(* Logix 5000 project; controller AdvManLab vendor 1 type 14 code 158 rev 28.12; software revision 28.01; part 9 of 13 *)
(* tags used below, declared in another part *)
   HMI_WritePart : DINT;
   ABB_Loop_Speed : DINT;
   Advance_Slide : BOOL;
   AutoDelay : TIMER;
   Cell1PalletAtStop : BOOL;   // Part at Cell 1 Pallet Stop
   Clamp_To_Line : BOOL;
   Close_Clamp : BOOL;
   CNC_1_Done : BOOL;   // CNC 1 has completed cutting the part
   CNC_2_Done : BOOL;   // CNC 2 has completed cutting the part
   Enable_Cell_3 : BOOL;   // Turn bit on to enable logic for Cell 3
   Enable_CNC1 : BOOL;
   Enable_CNC2 : BOOL;
   Enable_CNC3 : BOOL;
   Enable_CNC4 : BOOL;
   EnableBits : DINT;
   Extend_Stop : BOOL;
   Fanuc_Loop_Speed : DINT;
   Festo_Air_On : BOOL;
   FestoAI0 : DINT;
   FestoAI1 : DINT;
   FestoAI2 : DINT;
   FestoAI3 : DINT;
   FestoAIP0 : DINT;
   FestoAIP1 : DINT;
   FestoAIP2 : DINT;
   FestoAIP3 : DINT;
   Gantry_busy : BOOL;
   Gantry_prep : BOOL;
   Gantry_reload : BOOL;
   Gantry_start : BOOL;
   HMI_Disp_No : DINT;
   HMI_Mode : DINT;
   Lower_Slide : BOOL;
   Mode_Auto : BOOL;
   Mode_Manual : BOOL;
   Mode_None : BOOL;
   Mode_Semi : BOOL;
   Mode_Start : BOOL;
   NI_1752_Camera : MESSAGE;
   ONS : DINT;
   Open_Clamp : BOOL;
   PalletAtC2C3HoldBack : BOOL;   // Pallet at Cell 2 to Cell 3 Diverter Hold Back Stop
   Part_A : BOOL;
   Part_A_input : COUNTER;
   Part_A_output : COUNTER;
   Part_B : BOOL;
   Part_B_input : COUNTER;
   Part_B_output : COUNTER;
   Part_dropped : BOOL;
   Part_from_conv_holding : BOOL;
   Part_ready_for_Gantry : BOOL;
   Picking_up_part : BOOL;
   PPX4 : ALIAS FOR Conv_N053:3:I.2;   // Sensor Pallet Stop RFID4 (Loop 1 Diverter Hold Back Stop)
   PPX5 : ALIAS FOR Main_N043:3:I.0;   // Sensor Pallet Stop (Cell 1 Hold Back)
   R1J_Assign : BOOL;
   R1J_Check_Process_NO : DINT;
   R1J_Current_Part_NO : SINT;
   R1J_Current_Process_NO : SINT;
   R1J_Read : BOOL;
   R1J_Read_Check_Fail : BOOL;
   R1J_Read_Check_InProgress : BOOL;
   R1J_Read_Check_Results : BOOL;
   R1J_Read_Check_Start : BOOL;
   R1J_Read_Finished : BOOL;
   R1J_Read_InProgress : BOOL;
   R1J_Read_Results : BOOL;
   R1J_Read_Start : BOOL;
   R1J_Write : BOOL;
   R1J_Write_Finished_Check : BOOL;
   R1J_Write_Inprogress : BOOL;
   R1J_Write_Pass : BOOL;
   Raise_Slide : BOOL;
   Return_Slide : BOOL;
   RFID_ReadData5p : DINT;
   RFIDTP1 : ALIAS FOR RFID_N054:I.Channel[0].TagPresent;   // RFID Tag at Cell 1 Stop
   Robot1_DroppedP1 : BOOL;
   Robot1_DroppedP2 : BOOL;
   Robot1_Flipped : BOOL;
   Robot1DroppedPart : BOOL;
   Run_gantry_logic : BOOL;
   TimerG1 : TIMER;
   Vac_On : BOOL;
   Vac_To_Line : BOOL;
(* MainProgram, continued *)

ROUTINE Grantry_Logic_Prep   (* ladder *)
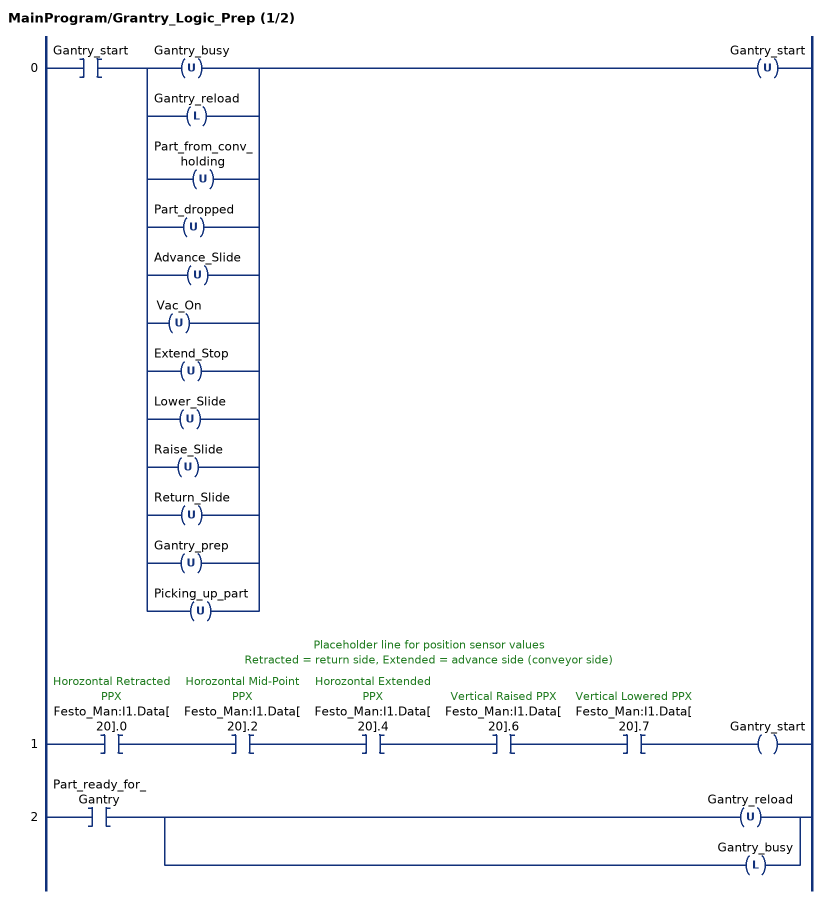
   0: XIC(Gantry_start)[OTU(Gantry_busy) ,OTL(Gantry_reload) ,OTU(Part_from_conv_holding) ,OTU(Part_dropped) ,OTU(Advance_Slide) ,OTU(Vac_On) ,OTU(Extend_Stop) ,OTU(Lower_Slide) ,OTU(Raise_Slide) ,OTU(Return_Slide) ,OTU(Gantry_prep) ,OTU(Picking_up_part) ]OTU(Gantry_start);
   // Placeholder line for position sensor values
   // Retracted = return side, Extended = advance side (conveyor side)
   1: XIC(Festo_Man:I1.Data[20].0)XIC(Festo_Man:I1.Data[20].2)XIC(Festo_Man:I1.Data[20].4)XIC(Festo_Man:I1.Data[20].6)XIC(Festo_Man:I1.Data[20].7)OTE(Gantry_start);
   2: XIC(Part_ready_for_Gantry)[OTU(Gantry_reload) ,OTL(Gantry_busy) ];
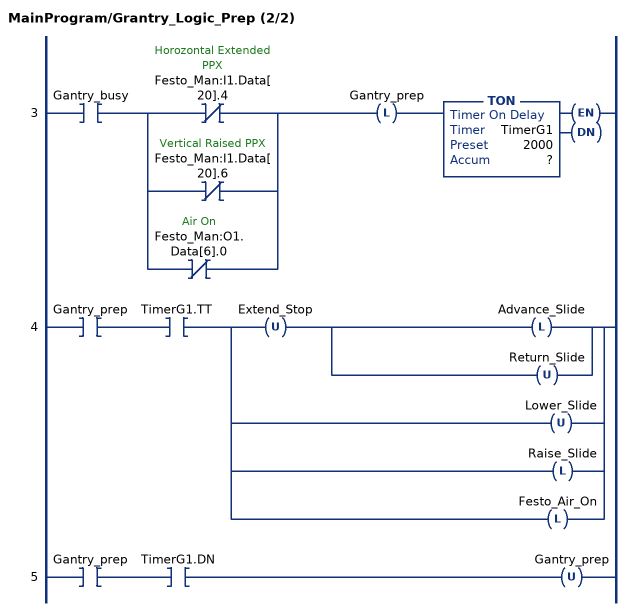
   3: XIC(Gantry_busy)[XIO(Festo_Man:I1.Data[20].4) ,XIO(Festo_Man:I1.Data[20].6) ,XIO(Festo_Man:O1.Data[6].0) ]OTL(Gantry_prep)TON(TimerG1,?,?);
   4: XIC(Gantry_prep)XIC(TimerG1.TT)[OTU(Extend_Stop) [OTL(Advance_Slide) ,OTU(Return_Slide) ] ,[OTU(Lower_Slide) ,OTL(Raise_Slide) ] ,OTL(Festo_Air_On) ];
   5: XIC(Gantry_prep)XIC(TimerG1.DN)OTU(Gantry_prep);
END_ROUTINE

ROUTINE HMI   (* ladder *)
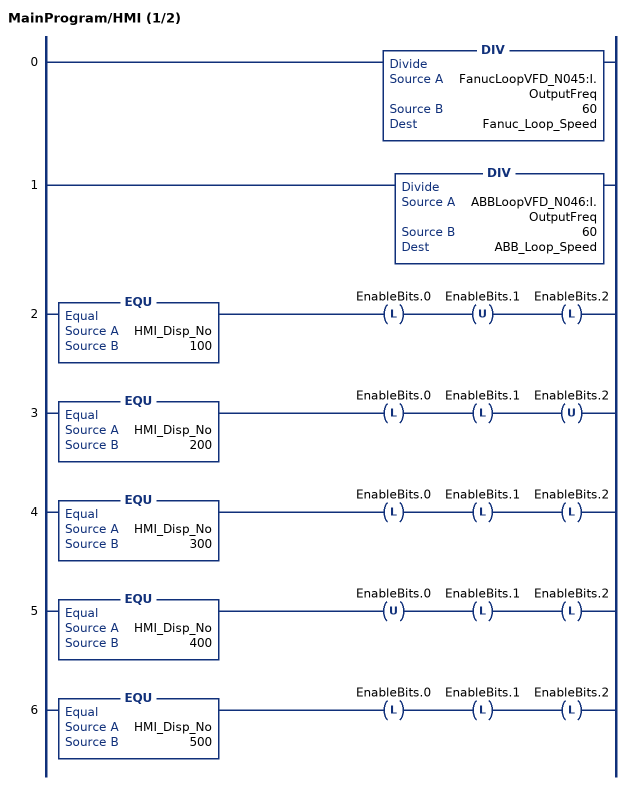
   0: DIV(FanucLoopVFD_N045:I.OutputFreq,60,Fanuc_Loop_Speed);
   1: DIV(ABBLoopVFD_N046:I.OutputFreq,60,ABB_Loop_Speed);
   2: EQU(HMI_Disp_No,100)OTL(EnableBits.0)OTU(EnableBits.1)OTL(EnableBits.2);
   3: EQU(HMI_Disp_No,200)OTL(EnableBits.0)OTL(EnableBits.1)OTU(EnableBits.2);
   4: EQU(HMI_Disp_No,300)OTL(EnableBits.0)OTL(EnableBits.1)OTL(EnableBits.2);
   5: EQU(HMI_Disp_No,400)OTU(EnableBits.0)OTL(EnableBits.1)OTL(EnableBits.2);
   6: EQU(HMI_Disp_No,500)OTL(EnableBits.0)OTL(EnableBits.1)OTL(EnableBits.2);
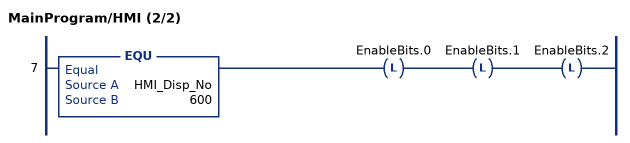
   7: EQU(HMI_Disp_No,600)OTL(EnableBits.0)OTL(EnableBits.1)OTL(EnableBits.2);
END_ROUTINE

ROUTINE MainRoutine   (* ladder *)
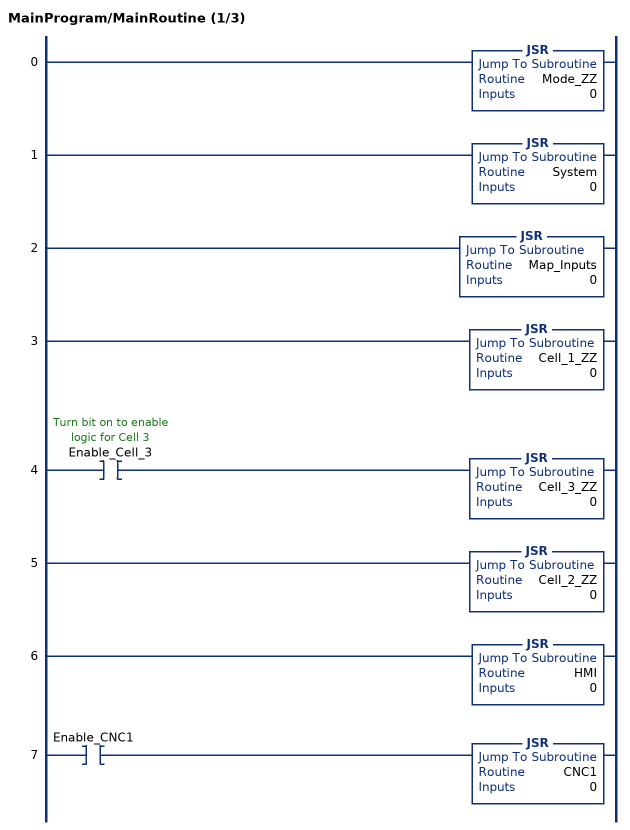
   0: JSR(Mode_ZZ,0);
   1: JSR(System,0);
   2: JSR(Map_Inputs,0);
   3: JSR(Cell_1_ZZ,0);
   4: XIC(Enable_Cell_3)JSR(Cell_3_ZZ,0);
   5: JSR(Cell_2_ZZ,0);
   6: JSR(HMI,0);
   7: XIC(Enable_CNC1)JSR(CNC1,0);
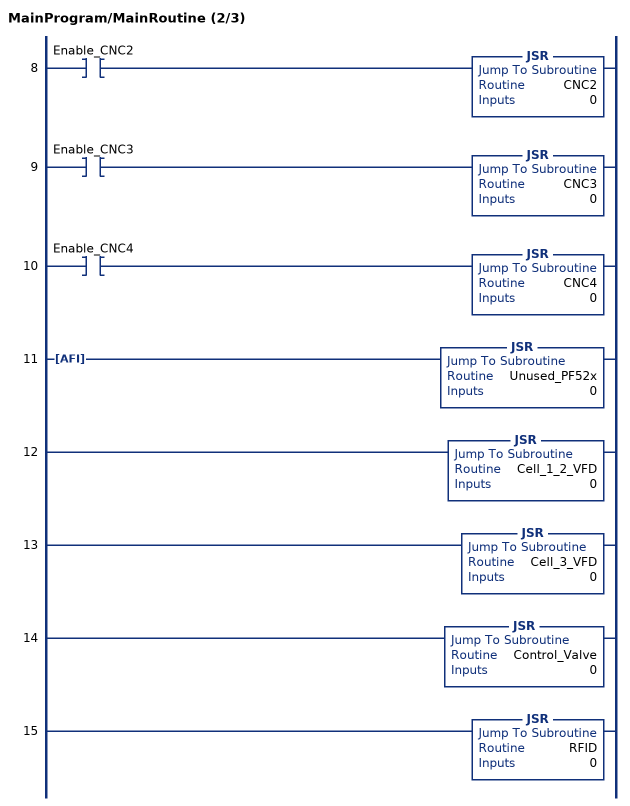
   8: XIC(Enable_CNC2)JSR(CNC2,0);
   9: XIC(Enable_CNC3)JSR(CNC3,0);
   10: XIC(Enable_CNC4)JSR(CNC4,0);
   11: AFI()JSR(Unused_PF52x,0);
   12: JSR(Cell_1_2_VFD,0);
   13: JSR(Cell_3_VFD,0);
   14: JSR(Control_Valve,0);
   15: JSR(RFID,0);
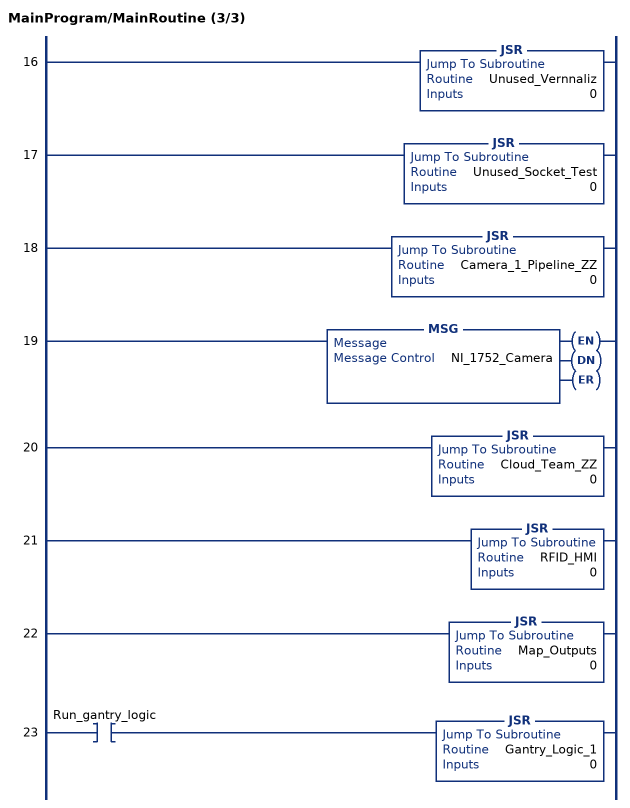
   16: JSR(Unused_Vernnaliz,0);
   17: JSR(Unused_Socket_Test,0);
   18: JSR(Camera_1_Pipeline_ZZ,0);
   19: MSG(NI_1752_Camera);
   20: JSR(Cloud_Team_ZZ,0);
   21: JSR(RFID_HMI,0);
   22: JSR(Map_Outputs,0);
   23: XIC(Run_gantry_logic)JSR(Gantry_Logic_1,0);
END_ROUTINE

ROUTINE Map_Inputs   (* ladder *)
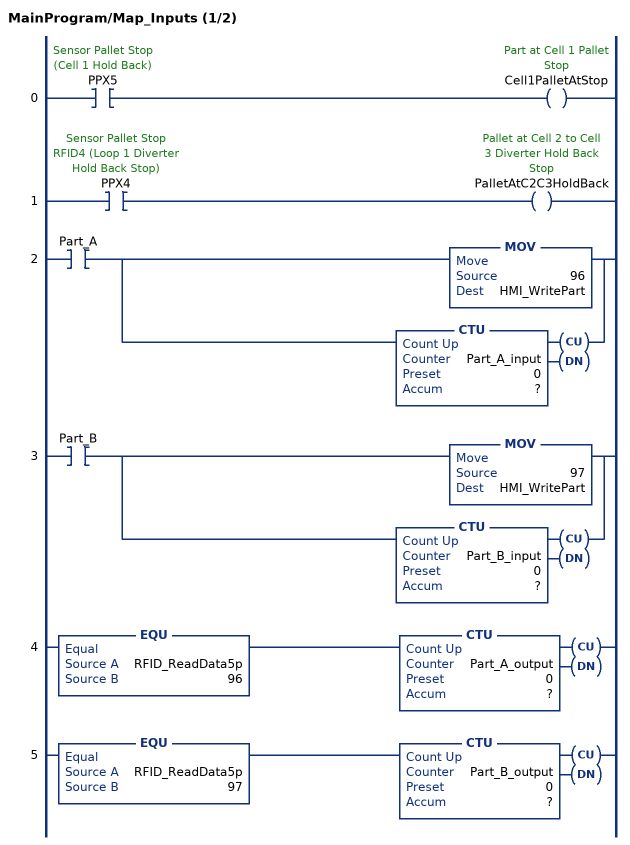
   0: XIC(PPX5)OTE(Cell1PalletAtStop);
   1: XIC(PPX4)OTE(PalletAtC2C3HoldBack);
   2: XIC(Part_A)[MOV(96,HMI_WritePart) ,CTU(Part_A_input,?,?) ];
   3: XIC(Part_B)[MOV(97,HMI_WritePart) ,CTU(Part_B_input,?,?) ];
   4: EQU(RFID_ReadData5p,96)CTU(Part_A_output,?,?);
   5: EQU(RFID_ReadData5p,97)CTU(Part_B_output,?,?);
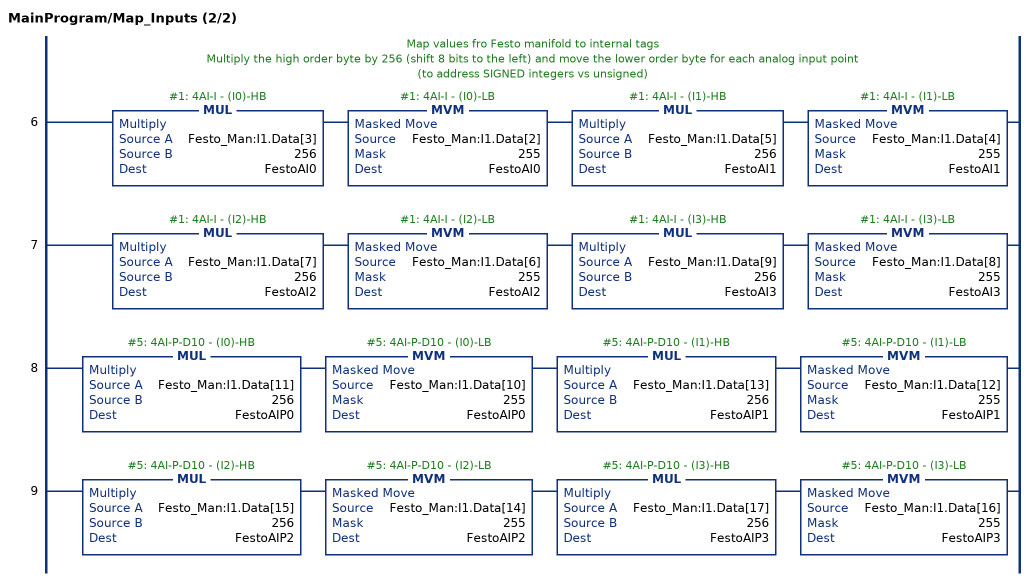
   // Map values fro Festo manifold to internal tags
   // Multiply the high order byte by 256 (shift 8 bits to the left) and move the lower order byte for each analog input point
   // (to address SIGNED integers vs unsigned)
   6: MUL(Festo_Man:I1.Data[3],256,FestoAI0)MVM(Festo_Man:I1.Data[2],255,FestoAI0)MUL(Festo_Man:I1.Data[5],256,FestoAI1)MVM(Festo_Man:I1.Data[4],255,FestoAI1);
   7: MUL(Festo_Man:I1.Data[7],256,FestoAI2)MVM(Festo_Man:I1.Data[6],255,FestoAI2)MUL(Festo_Man:I1.Data[9],256,FestoAI3)MVM(Festo_Man:I1.Data[8],255,FestoAI3);
   8: MUL(Festo_Man:I1.Data[11],256,FestoAIP0)MVM(Festo_Man:I1.Data[10],255,FestoAIP0)MUL(Festo_Man:I1.Data[13],256,FestoAIP1)MVM(Festo_Man:I1.Data[12],255,FestoAIP1);
   9: MUL(Festo_Man:I1.Data[15],256,FestoAIP2)MVM(Festo_Man:I1.Data[14],255,FestoAIP2)MUL(Festo_Man:I1.Data[17],256,FestoAIP3)MVM(Festo_Man:I1.Data[16],255,FestoAIP3);
END_ROUTINE

ROUTINE Map_Outputs   (* ladder *)
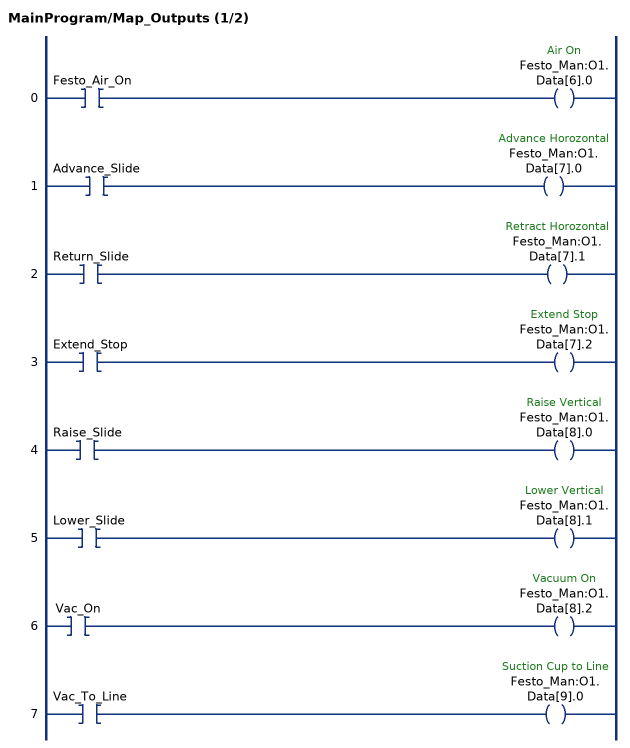
   0: XIC(Festo_Air_On)OTE(Festo_Man:O1.Data[6].0);
   1: XIC(Advance_Slide)OTE(Festo_Man:O1.Data[7].0);
   2: XIC(Return_Slide)OTE(Festo_Man:O1.Data[7].1);
   3: XIC(Extend_Stop)OTE(Festo_Man:O1.Data[7].2);
   4: XIC(Raise_Slide)OTE(Festo_Man:O1.Data[8].0);
   5: XIC(Lower_Slide)OTE(Festo_Man:O1.Data[8].1);
   6: XIC(Vac_On)OTE(Festo_Man:O1.Data[8].2);
   7: XIC(Vac_To_Line)OTE(Festo_Man:O1.Data[9].0);
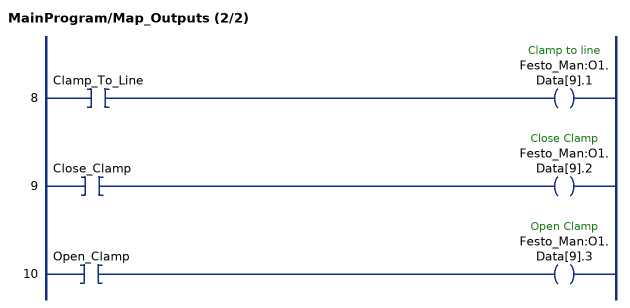
   8: XIC(Clamp_To_Line)OTE(Festo_Man:O1.Data[9].1);
   9: XIC(Close_Clamp)OTE(Festo_Man:O1.Data[9].2);
   10: XIC(Open_Clamp)OTE(Festo_Man:O1.Data[9].3);
END_ROUTINE

ROUTINE Mode_ZZ   (* ladder *)
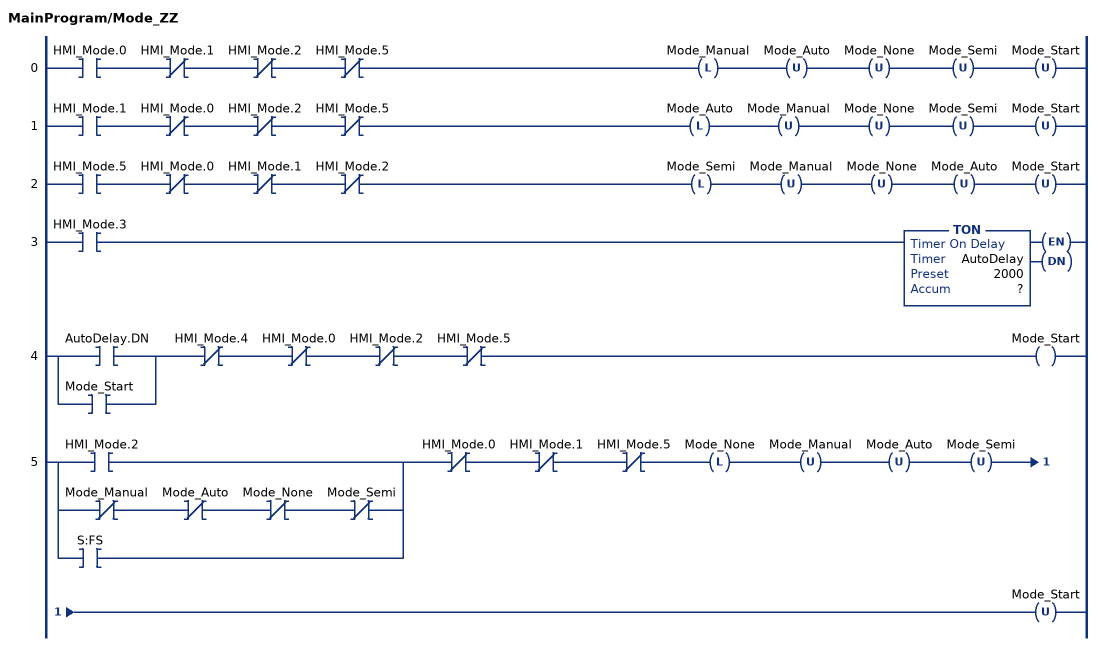
   0: XIC(HMI_Mode.0)XIO(HMI_Mode.1)XIO(HMI_Mode.2)XIO(HMI_Mode.5)OTL(Mode_Manual)OTU(Mode_Auto)OTU(Mode_None)OTU(Mode_Semi)OTU(Mode_Start);
   1: XIC(HMI_Mode.1)XIO(HMI_Mode.0)XIO(HMI_Mode.2)XIO(HMI_Mode.5)OTL(Mode_Auto)OTU(Mode_Manual)OTU(Mode_None)OTU(Mode_Semi)OTU(Mode_Start);
   2: XIC(HMI_Mode.5)XIO(HMI_Mode.0)XIO(HMI_Mode.1)XIO(HMI_Mode.2)OTL(Mode_Semi)OTU(Mode_Manual)OTU(Mode_None)OTU(Mode_Auto)OTU(Mode_Start);
   3: XIC(HMI_Mode.3)TON(AutoDelay,?,?);
   4: [XIC(AutoDelay.DN) ,XIC(Mode_Start) ]XIO(HMI_Mode.4)XIO(HMI_Mode.0)XIO(HMI_Mode.2)XIO(HMI_Mode.5)OTE(Mode_Start);
   5: [XIC(HMI_Mode.2) ,XIO(Mode_Manual) XIO(Mode_Auto) XIO(Mode_None) XIO(Mode_Semi) ,XIC(S:FS) ]XIO(HMI_Mode.0)XIO(HMI_Mode.1)XIO(HMI_Mode.5)OTL(Mode_None)OTU(Mode_Manual)OTU(Mode_Auto)OTU(Mode_Semi)OTU(Mode_Start);
END_ROUTINE

ROUTINE RFID   (* ladder *)
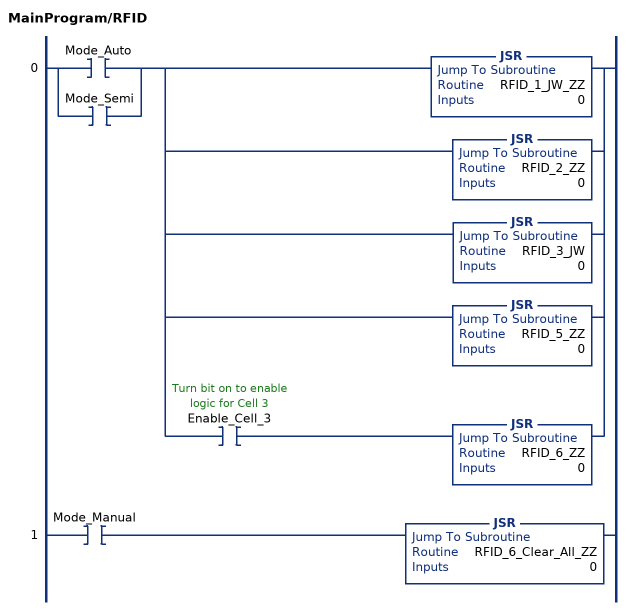
   0: [XIC(Mode_Auto) ,XIC(Mode_Semi) ][JSR(RFID_1_JW_ZZ,0) ,JSR(RFID_2_ZZ,0) ,JSR(RFID_3_JW,0) ,JSR(RFID_5_ZZ,0) ,XIC(Enable_Cell_3) JSR(RFID_6_ZZ,0) ];
   1: XIC(Mode_Manual)JSR(RFID_6_Clear_All_ZZ,0);
END_ROUTINE

ROUTINE RFID_1_JW_ZZ   (* ladder *)
// Rewrite of RFID_1 using new read/write logic of RFID_6_ZZ
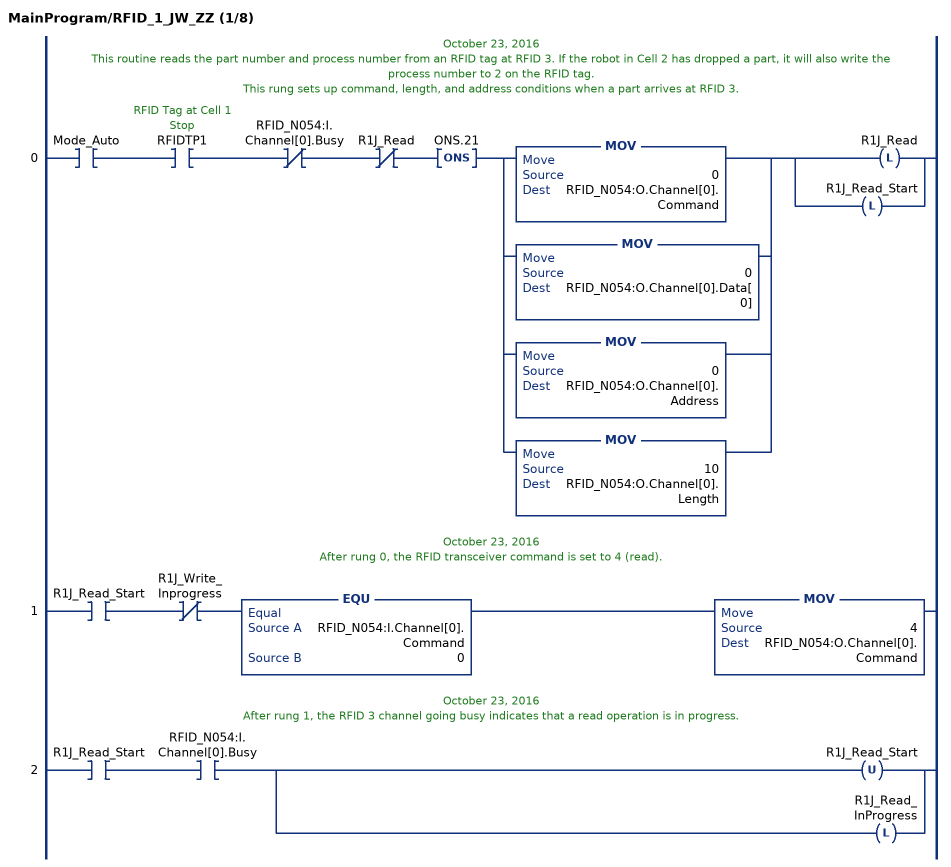
   // October 23, 2016
   // This routine reads the part number and process number from an RFID tag at RFID 3. If the robot in Cell 2 has dropped a part, it will also write the process number to 2 on the RFID tag.
   // This rung sets up command, length, and address conditions when a part arrives at RFID 3.
   0: XIC(Mode_Auto)XIC(RFIDTP1)XIO(RFID_N054:I.Channel[0].Busy)XIO(R1J_Read)ONS(ONS.21)[MOV(0,RFID_N054:O.Channel[0].Command) ,MOV(0,RFID_N054:O.Channel[0].Data[0]) ,MOV(0,RFID_N054:O.Channel[0].Address) ,MOV(10,RFID_N054:O.Channel[0].Length) ][OTL(R1J_Read) ,OTL(R1J_Read_Start) ];
   // October 23, 2016
   // After rung 0, the RFID transceiver command is set to 4 (read).
   1: XIC(R1J_Read_Start)XIO(R1J_Write_Inprogress)EQU(RFID_N054:I.Channel[0].Command,0)MOV(4,RFID_N054:O.Channel[0].Command);
   // October 23, 2016
   // After rung 1, the RFID 3 channel going busy indicates that a read operation is in progress.
   2: XIC(R1J_Read_Start)XIC(RFID_N054:I.Channel[0].Busy)[OTU(R1J_Read_Start) ,OTL(R1J_Read_InProgress) ];
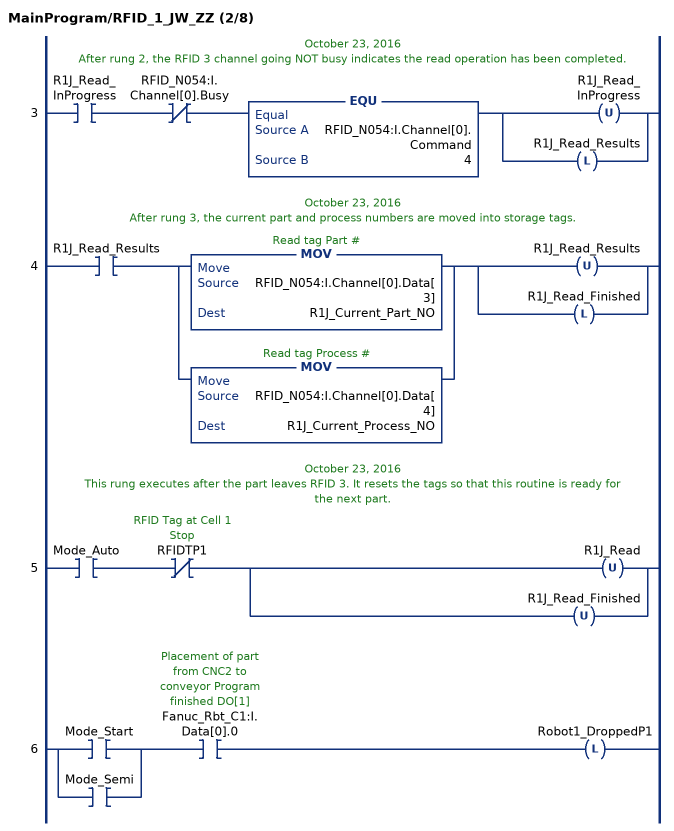
   // October 23, 2016
   // After rung 2, the RFID 3 channel going NOT busy indicates the read operation has been completed.
   3: XIC(R1J_Read_InProgress)XIO(RFID_N054:I.Channel[0].Busy)EQU(RFID_N054:I.Channel[0].Command,4)[OTU(R1J_Read_InProgress) ,OTL(R1J_Read_Results) ];
   // October 23, 2016
   // After rung 3, the current part and process numbers are moved into storage tags.
   4: XIC(R1J_Read_Results)[MOV(RFID_N054:I.Channel[0].Data[3],R1J_Current_Part_NO) ,MOV(RFID_N054:I.Channel[0].Data[4],R1J_Current_Process_NO) ][OTU(R1J_Read_Results) ,OTL(R1J_Read_Finished) ];
   // October 23, 2016
   // This rung executes after the part leaves RFID 3. It resets the tags so that this routine is ready for the next part.
   5: XIC(Mode_Auto)XIO(RFIDTP1)[OTU(R1J_Read) ,OTU(R1J_Read_Finished) ];
   6: [XIC(Mode_Start) ,XIC(Mode_Semi) ]XIC(Fanuc_Rbt_C1:I.Data[0].0)OTL(Robot1_DroppedP1);
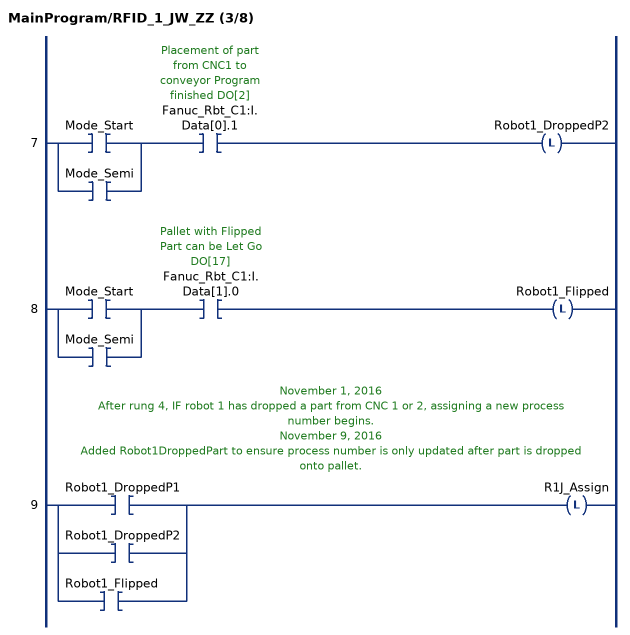
   7: [XIC(Mode_Start) ,XIC(Mode_Semi) ]XIC(Fanuc_Rbt_C1:I.Data[0].1)OTL(Robot1_DroppedP2);
   8: [XIC(Mode_Start) ,XIC(Mode_Semi) ]XIC(Fanuc_Rbt_C1:I.Data[1].0)OTL(Robot1_Flipped);
   // November 1, 2016
   // After rung 4, IF robot 1 has dropped a part from CNC 1 or 2, assigning a new process number begins.
   // November 9, 2016
   // Added Robot1DroppedPart to ensure process number is only updated after part is dropped onto pallet.
   9: [XIC(Robot1_DroppedP1) ,XIC(Robot1_DroppedP2) ,XIC(Robot1_Flipped) ]OTL(R1J_Assign);
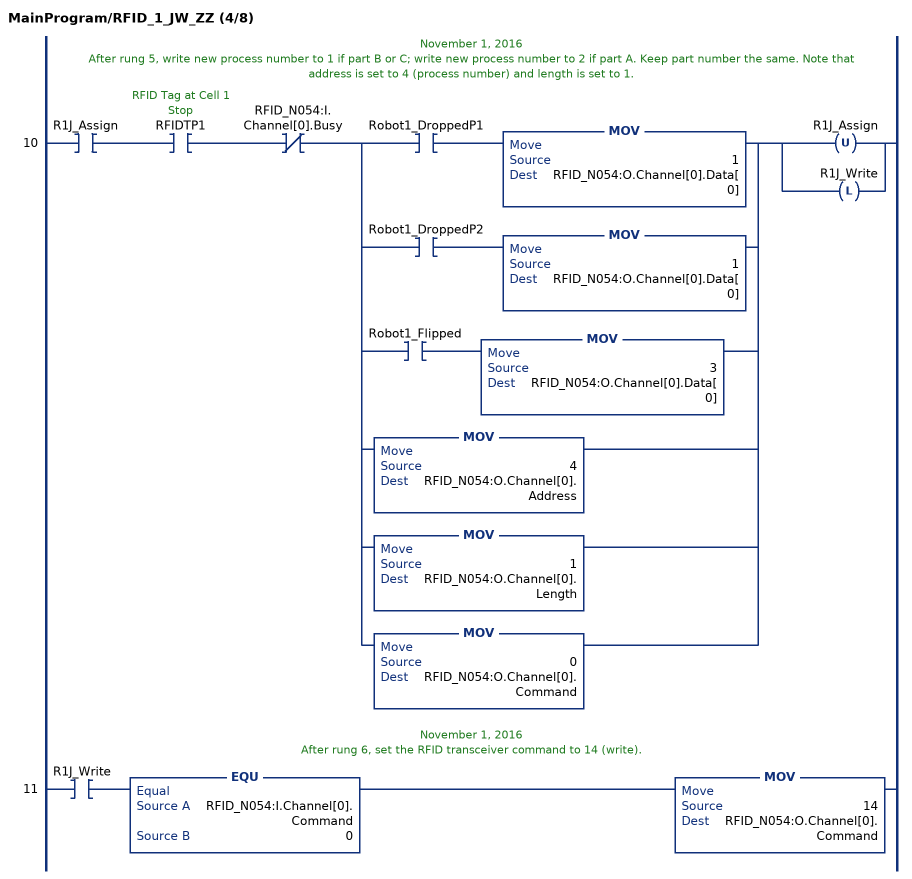
   // November 1, 2016
   // After rung 5, write new process number to 1 if part B or C; write new process number to 2 if part A. Keep part number the same. Note that address is set to 4 (process number) and length is set to 1.
   10: XIC(R1J_Assign)XIC(RFIDTP1)XIO(RFID_N054:I.Channel[0].Busy)[XIC(Robot1_DroppedP1) MOV(1,RFID_N054:O.Channel[0].Data[0]) ,XIC(Robot1_DroppedP2) MOV(1,RFID_N054:O.Channel[0].Data[0]) ,XIC(Robot1_Flipped) MOV(3,RFID_N054:O.Channel[0].Data[0]) ,MOV(4,RFID_N054:O.Channel[0].Address) ,MOV(1,RFID_N054:O.Channel[0].Length) ,MOV(0,RFID_N054:O.Channel[0].Command) ][OTU(R1J_Assign) ,OTL(R1J_Write) ];
   // November 1, 2016
   // After rung 6, set the RFID transceiver command to 14 (write).
   11: XIC(R1J_Write)EQU(RFID_N054:I.Channel[0].Command,0)MOV(14,RFID_N054:O.Channel[0].Command);
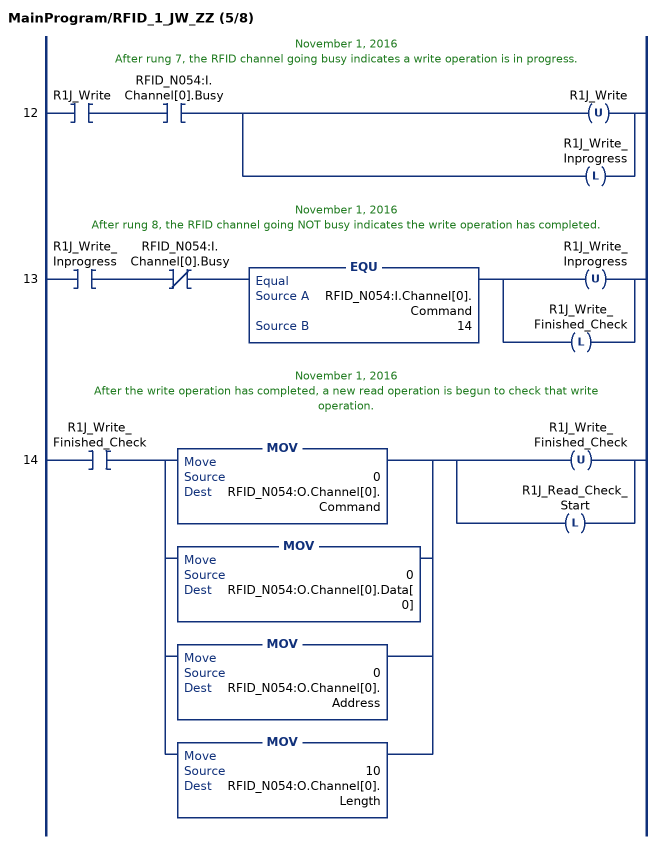
   // November 1, 2016
   // After rung 7, the RFID channel going busy indicates a write operation is in progress.
   12: XIC(R1J_Write)XIC(RFID_N054:I.Channel[0].Busy)[OTU(R1J_Write) ,OTL(R1J_Write_Inprogress) ];
   // November 1, 2016
   // After rung 8, the RFID channel going NOT busy indicates the write operation has completed.
   13: XIC(R1J_Write_Inprogress)XIO(RFID_N054:I.Channel[0].Busy)EQU(RFID_N054:I.Channel[0].Command,14)[OTU(R1J_Write_Inprogress) ,OTL(R1J_Write_Finished_Check) ];
   // November 1, 2016
   // After the write operation has completed, a new read operation is begun to check that write operation.
   14: XIC(R1J_Write_Finished_Check)[MOV(0,RFID_N054:O.Channel[0].Command) ,MOV(0,RFID_N054:O.Channel[0].Data[0]) ,MOV(0,RFID_N054:O.Channel[0].Address) ,MOV(10,RFID_N054:O.Channel[0].Length) ][OTU(R1J_Write_Finished_Check) ,OTL(R1J_Read_Check_Start) ];
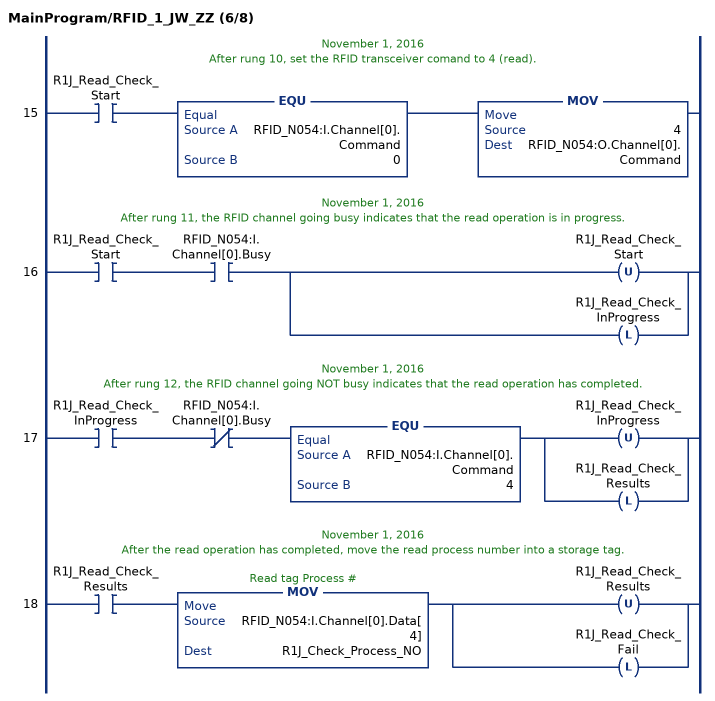
   // November 1, 2016
   // After rung 10, set the RFID transceiver comand to 4 (read).
   15: XIC(R1J_Read_Check_Start)EQU(RFID_N054:I.Channel[0].Command,0)MOV(4,RFID_N054:O.Channel[0].Command);
   // November 1, 2016
   // After rung 11, the RFID channel going busy indicates that the read operation is in progress.
   16: XIC(R1J_Read_Check_Start)XIC(RFID_N054:I.Channel[0].Busy)[OTU(R1J_Read_Check_Start) ,OTL(R1J_Read_Check_InProgress) ];
   // November 1, 2016
   // After rung 12, the RFID channel going NOT busy indicates that the read operation has completed.
   17: XIC(R1J_Read_Check_InProgress)XIO(RFID_N054:I.Channel[0].Busy)EQU(RFID_N054:I.Channel[0].Command,4)[OTU(R1J_Read_Check_InProgress) ,OTL(R1J_Read_Check_Results) ];
   // November 1, 2016
   // After the read operation has completed, move the read process number into a storage tag.
   18: XIC(R1J_Read_Check_Results)MOV(RFID_N054:I.Channel[0].Data[4],R1J_Check_Process_NO)[OTU(R1J_Read_Check_Results) ,OTL(R1J_Read_Check_Fail) ];
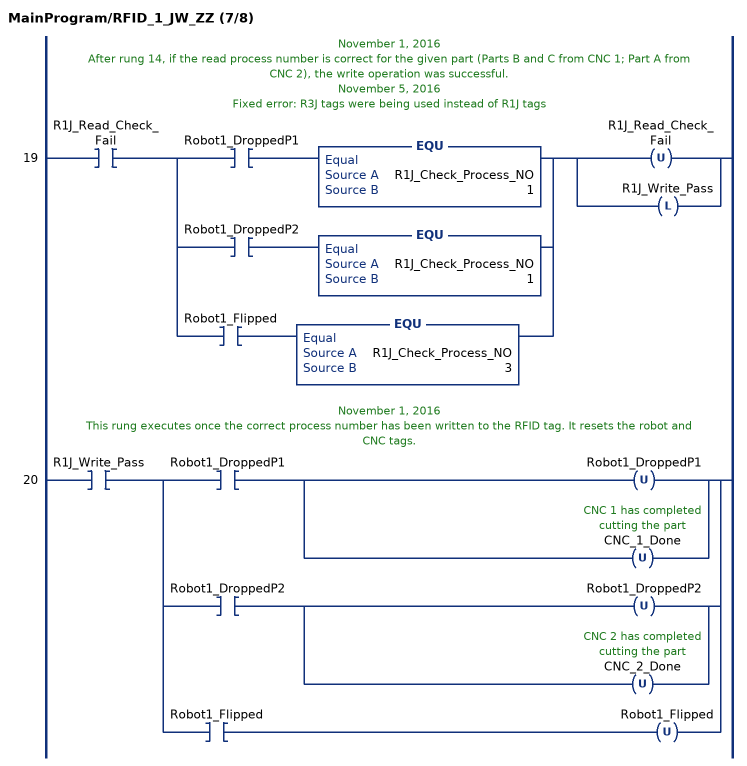
   // November 1, 2016
   // After rung 14, if the read process number is correct for the given part (Parts B and C from CNC 1; Part A from CNC 2), the write operation was successful.
   // November 5, 2016
   // Fixed error: R3J tags were being used instead of R1J tags
   19: XIC(R1J_Read_Check_Fail)[XIC(Robot1_DroppedP1) EQU(R1J_Check_Process_NO,1) ,XIC(Robot1_DroppedP2) EQU(R1J_Check_Process_NO,1) ,XIC(Robot1_Flipped) EQU(R1J_Check_Process_NO,3) ][OTU(R1J_Read_Check_Fail) ,OTL(R1J_Write_Pass) ];
   // November 1, 2016
   // This rung executes once the correct process number has been written to the RFID tag. It resets the robot and CNC tags.
   20: XIC(R1J_Write_Pass)[XIC(Robot1_DroppedP1) [OTU(Robot1_DroppedP1) ,OTU(CNC_1_Done) ] ,XIC(Robot1_DroppedP2) [OTU(Robot1_DroppedP2) ,OTU(CNC_2_Done) ] ,XIC(Robot1_Flipped) OTU(Robot1_Flipped) ];
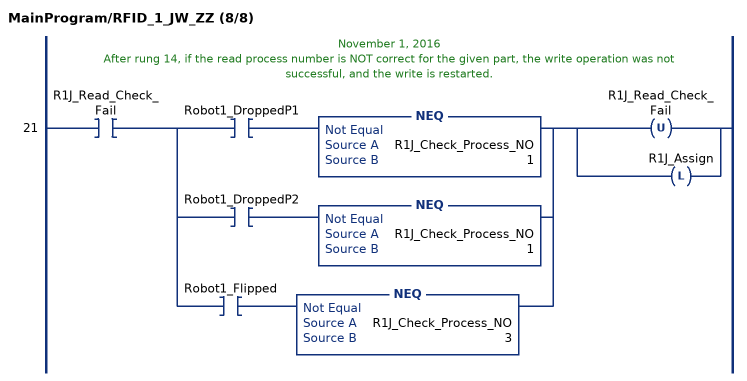
   // November 1, 2016
   // After rung 14, if the read process number is NOT correct for the given part, the write operation was not successful, and the write is restarted.
   21: XIC(R1J_Read_Check_Fail)[XIC(Robot1_DroppedP1) NEQ(R1J_Check_Process_NO,1) ,XIC(Robot1_DroppedP2) NEQ(R1J_Check_Process_NO,1) ,XIC(Robot1_Flipped) NEQ(R1J_Check_Process_NO,3) ][OTU(R1J_Read_Check_Fail) ,OTL(R1J_Assign) ];
END_ROUTINE
